SYSTEM xghhx
  (* Version 1.0, 2022-05-13, admin *)
  APPLICATION xghhxApp
    FBS
      E_RESTART : E_RESTART;
      E_PERMIT : E_PERMIT(PERMIT := 1);
      E_PERMIT_1 : E_PERMIT;
    END_FBS
    EVENT_CONNECTIONS
      E_RESTART.WARM TO E_PERMIT.EI;
      E_PERMIT.EO TO E_PERMIT_1.EI;
    END_CONNECTIONS
  END_APPLICATION
END_SYSTEM
